(*
SPDX-FileCopyrightText: © 2026 Oleksandr Tiutyk <trofimich@gmail.com>
SPDX-License-Identifier: MIT
License: https://opensource.org/license/mit
*)

INTERFACE IStandardException EXTENDS IGeneralException

METHOD Throw
VAR_INPUT
	sourceNamespaceName : STRING;
	sourceClassName : STRING;
	sourcePOUName : STRING;
	sourcePosition : STRING;
	message : ERROR_MESSAGE;
	errorCode : UDINT := 0;
	innerException : IException := 0;
END_VAR
END_METHOD

END_INTERFACE

(* stored: Version 1.1.0.1
   Itf IStandardException: Id {44bc1fac-e5a7-4db5-b697-c8ac44e9b553}
   Method Throw: Id {2a459ebf-4fc3-4850-993f-95d325724c5e} *)
